// TIA Portal V20 export
TYPE "MABS"
// stored: Access Published, Namespace LineD1
   STRUCT
      Run_balls : Bool := false;   // Run transport balls
      Dir_balls : Bool := false;   // 0=forward; 1=backward
      Speed_balls : Int := 90;   // Based on preset speed setting. 60/70/80/90 m/min.
      Switch_left_angle : Int := 45;   // Angle for left transportation 30/180°
      Switch_right_angle : Int := 45;   // Angle for right transportation 30/180°
      Switch_left_to_st_offset : Int := 0;   // Offset angle for straight position from left -8/+10°
      Switch_right_to_st_offset : Int := 0;   // Offset angle for straight position from right -8/+10°
      Init_offset : Int := 0;   // Offset angle for initial position -8/+10°
      Switch_left : Bool := false;   // Swing to left transport direction
      Switch_right : Bool := false;   // Swing to right transport direction
      Switch_left_to_st : Bool := false;   // Swing to straight transport direction CW
      Switch_right_to_st : Bool := false;   // Swing to straight transport direction CCW
      EMS : Bool := false;   // Inhib controls and reset MABS initialisation
      Init : Bool := false;   // Run MABS initialisation sequence (if not done)
      Init_done : Bool := false;   // MABS initialisation sequence done
      Ready : Bool := false;   // MABS no error, initialisation done, communication OK
      Init_sensor : Bool := false;   // MABS straight position sensor
      Left_Pos_reach : Bool := false;   // MABS transport balls in left position
      Right_Pos_reach : Bool := false;   // MABS transport balls in right position
      Straight_Pos_reach : Bool := false;   // MABS transport balls in straight position
      Error_motA : Bool := false;   // Hardware error motor A
      Error_motB : Bool := false;   // Hardware error motor B
      Error_timeout_sw : Bool := false;   // Swing motor timeout
      Error_com : Bool := false;   // Communication error (life bit, 5s delayed)
      Error : Bool := false;   // Error synthesis
      Reset_error : Bool := false;   // Reset all errors
      Timeout_val : Time := T#10s;   // Swing timeout value
      HMI_sts : UInt := 0;   // Sts word for HMI (0=Off; 1=Running; 2=Init requested; 4=Error )
   END_STRUCT;
END_TYPE
